Xinje XCPPro project, PLC1: XC2-32 (software 3.3r 2017-11-24)

PROGRAM Ladder

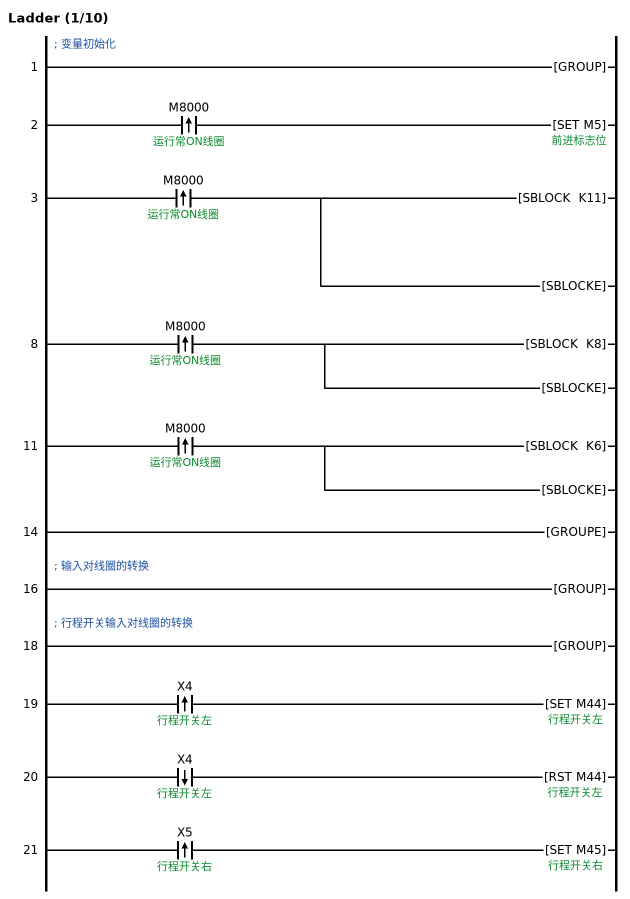
; 变量初始化
GROUP
LDP    M8000	; 运行常ON线圈
SET    M5	; 前进标志位
LDP    M8000	; 运行常ON线圈
SBLOCK K11
SBLOCKE
LDP    M8000	; 运行常ON线圈
SBLOCK K8
SBLOCKE
LDP    M8000	; 运行常ON线圈
SBLOCK K6
SBLOCKE
GROUPE
; 输入对线圈的转换
GROUP
; 行程开关输入对线圈的转换
GROUP
LDP    X4	; 行程开关左
SET    M44	; 行程开关左
LDF    X4	; 行程开关左
RST    M44	; 行程开关左
LDP    X5	; 行程开关右
SET    M45	; 行程开关右

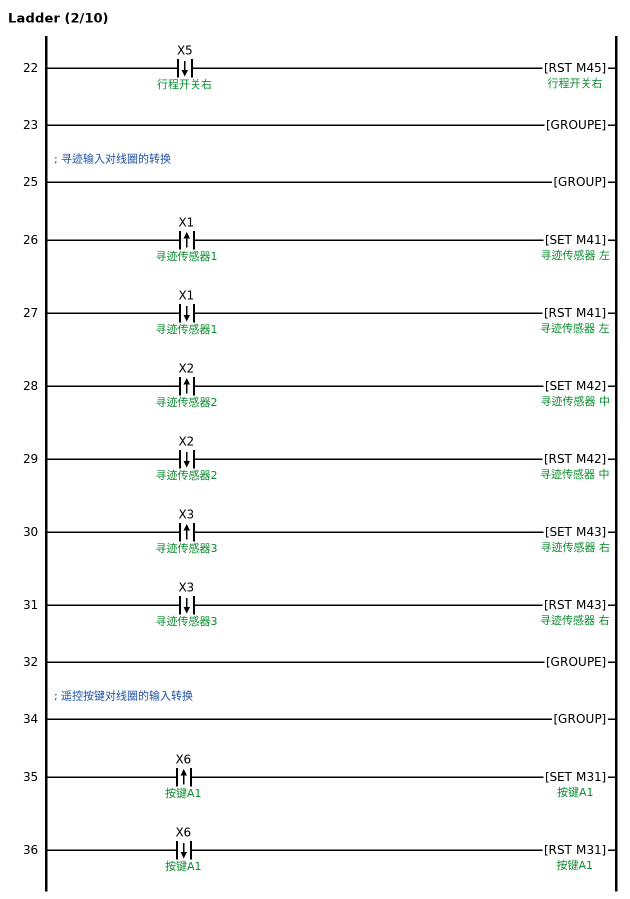
LDF    X5	; 行程开关右
RST    M45	; 行程开关右
GROUPE
; 寻迹输入对线圈的转换
GROUP
LDP    X1	; 寻迹传感器1
SET    M41	; 寻迹传感器 左
LDF    X1	; 寻迹传感器1
RST    M41	; 寻迹传感器 左
LDP    X2	; 寻迹传感器2
SET    M42	; 寻迹传感器 中
LDF    X2	; 寻迹传感器2
RST    M42	; 寻迹传感器 中
LDP    X3	; 寻迹传感器3
SET    M43	; 寻迹传感器 右
LDF    X3	; 寻迹传感器3
RST    M43	; 寻迹传感器 右
GROUPE
; 遥控按键对线圈的输入转换
GROUP
LDP    X6	; 按键A1
SET    M31	; 按键A1
LDF    X6	; 按键A1
RST    M31	; 按键A1

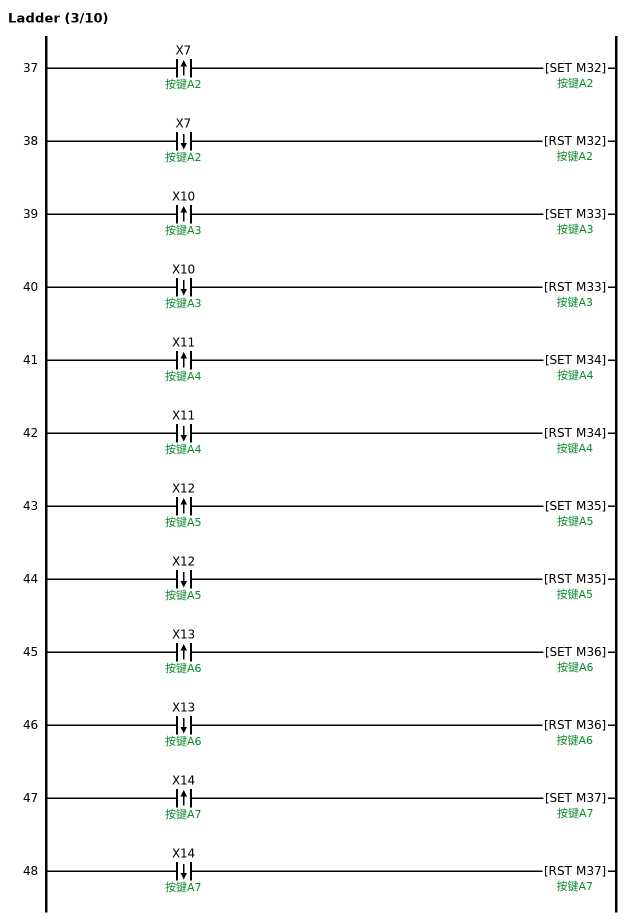
LDP    X7	; 按键A2
SET    M32	; 按键A2
LDF    X7	; 按键A2
RST    M32	; 按键A2
LDP    X10	; 按键A3
SET    M33	; 按键A3
LDF    X10	; 按键A3
RST    M33	; 按键A3
LDP    X11	; 按键A4
SET    M34	; 按键A4
LDF    X11	; 按键A4
RST    M34	; 按键A4
LDP    X12	; 按键A5
SET    M35	; 按键A5
LDF    X12	; 按键A5
RST    M35	; 按键A5
LDP    X13	; 按键A6
SET    M36	; 按键A6
LDF    X13	; 按键A6
RST    M36	; 按键A6
LDP    X14	; 按键A7
SET    M37	; 按键A7
LDF    X14	; 按键A7
RST    M37	; 按键A7

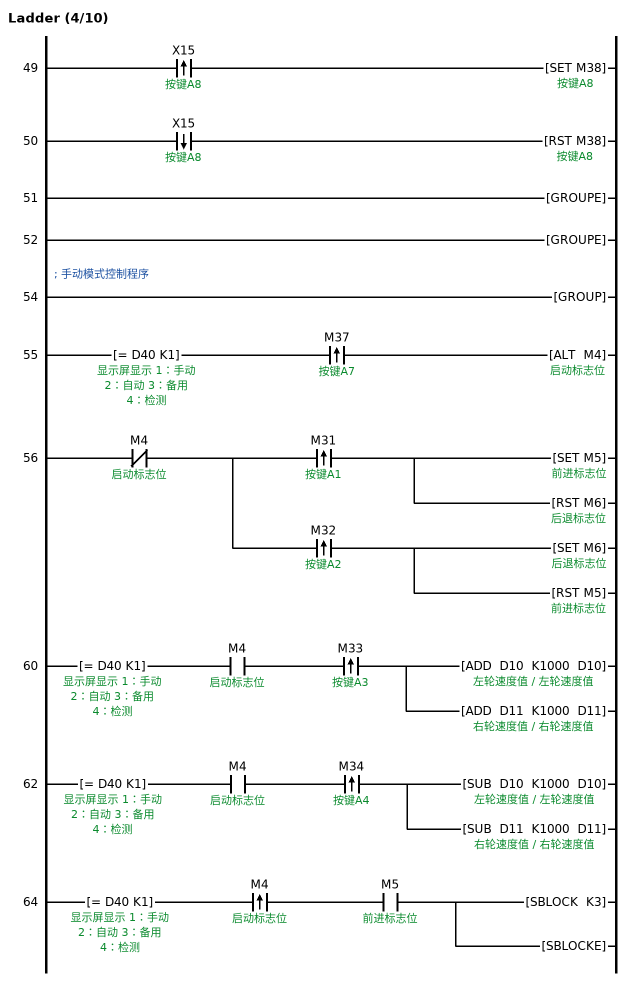
LDP    X15	; 按键A8
SET    M38	; 按键A8
LDF    X15	; 按键A8
RST    M38	; 按键A8
GROUPE
GROUPE
; 手动模式控制程序
GROUP
LD=    D40 K1	; 显示屏显示 1：手动 2：自动 3：备用 4：检测
ANDP   M37	; 按键A7
ALT    M4	; 启动标志位
LDI    M4	; 启动标志位
MPS
ANDP   M31	; 按键A1
SET    M5	; 前进标志位
RST    M6	; 后退标志位
MPP
ANDP   M32	; 按键A2
SET    M6	; 后退标志位
RST    M5	; 前进标志位
LD=    D40 K1	; 显示屏显示 1：手动 2：自动 3：备用 4：检测
AND    M4	; 启动标志位
ANDP   M33	; 按键A3
ADD    D10 K1000 D10	; 左轮速度值 / 左轮速度值
ADD    D11 K1000 D11	; 右轮速度值 / 右轮速度值
LD=    D40 K1	; 显示屏显示 1：手动 2：自动 3：备用 4：检测
AND    M4	; 启动标志位
ANDP   M34	; 按键A4
SUB    D10 K1000 D10	; 左轮速度值 / 左轮速度值
SUB    D11 K1000 D11	; 右轮速度值 / 右轮速度值
LD=    D40 K1	; 显示屏显示 1：手动 2：自动 3：备用 4：检测
ANDP   M4	; 启动标志位
AND    M5	; 前进标志位
SBLOCK K3
SBLOCKE

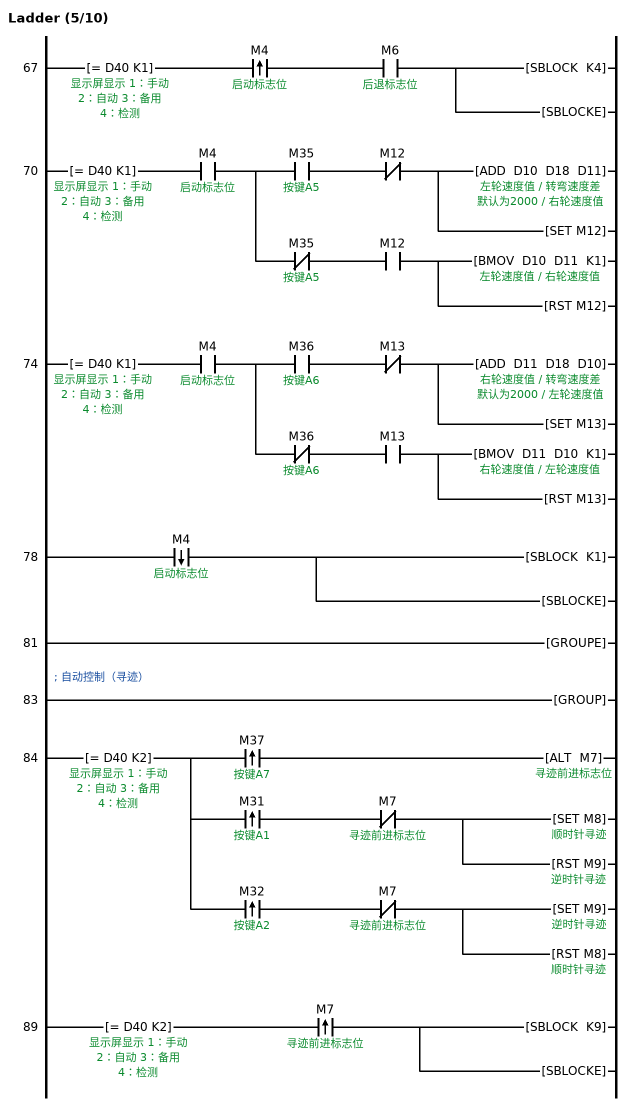
LD=    D40 K1	; 显示屏显示 1：手动 2：自动 3：备用 4：检测
ANDP   M4	; 启动标志位
AND    M6	; 后退标志位
SBLOCK K4
SBLOCKE
LD=    D40 K1	; 显示屏显示 1：手动 2：自动 3：备用 4：检测
AND    M4	; 启动标志位
MPS
AND    M35	; 按键A5
ANI    M12
ADD    D10 D18 D11	; 左轮速度值 / 转弯速度差 默认为2000 / 右轮速度值
SET    M12
MPP
ANI    M35	; 按键A5
AND    M12
BMOV   D10 D11 K1	; 左轮速度值 / 右轮速度值
RST    M12
LD=    D40 K1	; 显示屏显示 1：手动 2：自动 3：备用 4：检测
AND    M4	; 启动标志位
MPS
AND    M36	; 按键A6
ANI    M13
ADD    D11 D18 D10	; 右轮速度值 / 转弯速度差 默认为2000 / 左轮速度值
SET    M13
MPP
ANI    M36	; 按键A6
AND    M13
BMOV   D11 D10 K1	; 右轮速度值 / 左轮速度值
RST    M13
LDF    M4	; 启动标志位
SBLOCK K1
SBLOCKE
GROUPE
; 自动控制（寻迹）
GROUP
LD=    D40 K2	; 显示屏显示 1：手动 2：自动 3：备用 4：检测
MPS
ANDP   M37	; 按键A7
ALT    M7	; 寻迹前进标志位
MRD
ANDP   M31	; 按键A1
ANI    M7	; 寻迹前进标志位
SET    M8	; 顺时针寻迹
RST    M9	; 逆时针寻迹
MPP
ANDP   M32	; 按键A2
ANI    M7	; 寻迹前进标志位
SET    M9	; 逆时针寻迹
RST    M8	; 顺时针寻迹
LD=    D40 K2	; 显示屏显示 1：手动 2：自动 3：备用 4：检测
ANDP   M7	; 寻迹前进标志位
SBLOCK K9
SBLOCKE

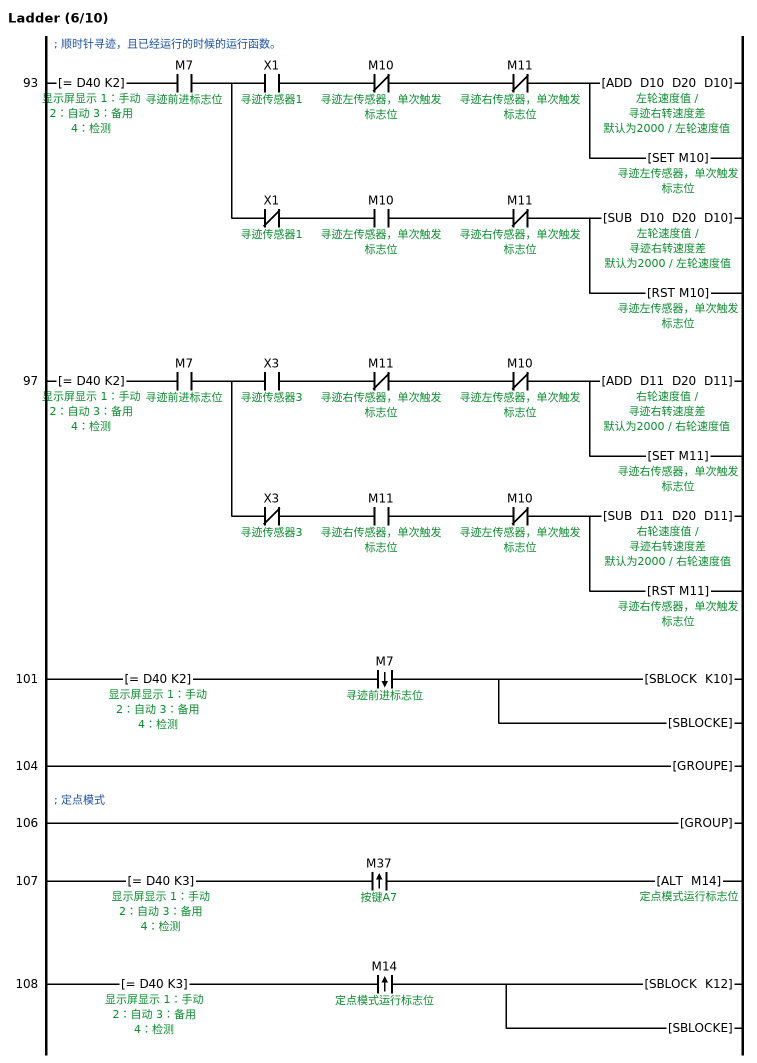
; 顺时针寻迹，且已经运行的时候的运行函数。
LD=    D40 K2	; 显示屏显示 1：手动 2：自动 3：备用 4：检测
AND    M7	; 寻迹前进标志位
MPS
AND    X1	; 寻迹传感器1
ANI    M10	; 寻迹左传感器，单次触发标志位
ANI    M11	; 寻迹右传感器，单次触发标志位
ADD    D10 D20 D10	; 左轮速度值 / 寻迹右转速度差 默认为2000 / 左轮速度值
SET    M10	; 寻迹左传感器，单次触发标志位
MPP
ANI    X1	; 寻迹传感器1
AND    M10	; 寻迹左传感器，单次触发标志位
ANI    M11	; 寻迹右传感器，单次触发标志位
SUB    D10 D20 D10	; 左轮速度值 / 寻迹右转速度差 默认为2000 / 左轮速度值
RST    M10	; 寻迹左传感器，单次触发标志位
LD=    D40 K2	; 显示屏显示 1：手动 2：自动 3：备用 4：检测
AND    M7	; 寻迹前进标志位
MPS
AND    X3	; 寻迹传感器3
ANI    M11	; 寻迹右传感器，单次触发标志位
ANI    M10	; 寻迹左传感器，单次触发标志位
ADD    D11 D20 D11	; 右轮速度值 / 寻迹右转速度差 默认为2000 / 右轮速度值
SET    M11	; 寻迹右传感器，单次触发标志位
MPP
ANI    X3	; 寻迹传感器3
AND    M11	; 寻迹右传感器，单次触发标志位
ANI    M10	; 寻迹左传感器，单次触发标志位
SUB    D11 D20 D11	; 右轮速度值 / 寻迹右转速度差 默认为2000 / 右轮速度值
RST    M11	; 寻迹右传感器，单次触发标志位
LD=    D40 K2	; 显示屏显示 1：手动 2：自动 3：备用 4：检测
ANDF   M7	; 寻迹前进标志位
SBLOCK K10
SBLOCKE
GROUPE
; 定点模式
GROUP
LD=    D40 K3	; 显示屏显示 1：手动 2：自动 3：备用 4：检测
ANDP   M37	; 按键A7
ALT    M14	; 定点模式运行标志位
LD=    D40 K3	; 显示屏显示 1：手动 2：自动 3：备用 4：检测
ANDP   M14	; 定点模式运行标志位
SBLOCK K12
SBLOCKE

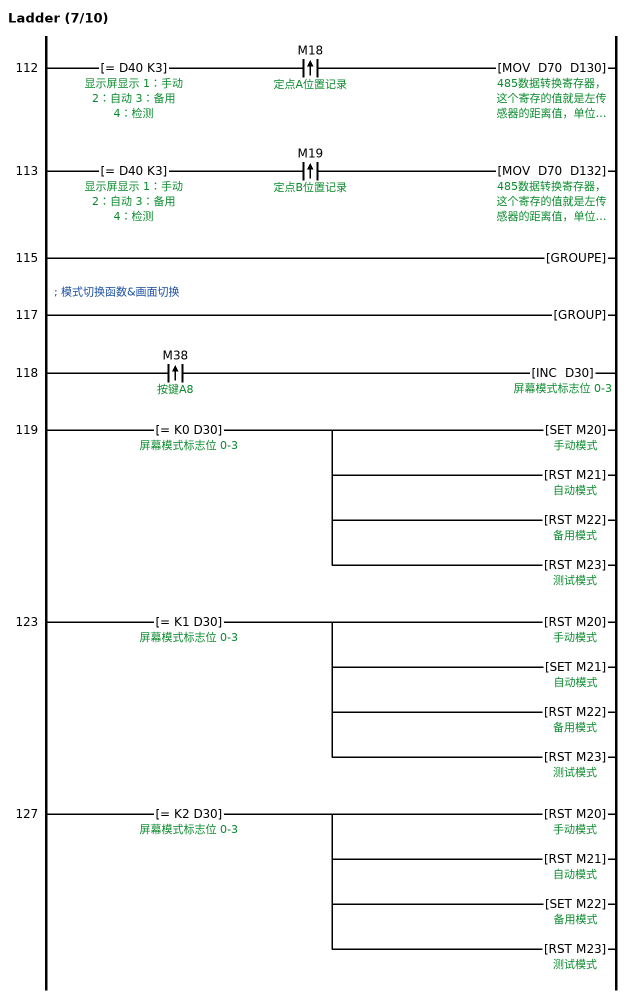
LD=    D40 K3	; 显示屏显示 1：手动 2：自动 3：备用 4：检测
ANDP   M18	; 定点A位置记录
MOV    D70 D130	; 485数据转换寄存器，这个寄存的值就是左传感器的距离值，单位mm / 定点模式A与墙面的距离
LD=    D40 K3	; 显示屏显示 1：手动 2：自动 3：备用 4：检测
ANDP   M19	; 定点B位置记录
MOV    D70 D132	; 485数据转换寄存器，这个寄存的值就是左传感器的距离值，单位mm / 定点模式B与墙面的距离
GROUPE
; 模式切换函数&画面切换
GROUP
LDP    M38	; 按键A8
INC    D30	; 屏幕模式标志位 0-3
LD=    K0 D30	; 屏幕模式标志位 0-3
SET    M20	; 手动模式
RST    M21	; 自动模式
RST    M22	; 备用模式
RST    M23	; 测试模式
LD=    K1 D30	; 屏幕模式标志位 0-3
RST    M20	; 手动模式
SET    M21	; 自动模式
RST    M22	; 备用模式
RST    M23	; 测试模式
LD=    K2 D30	; 屏幕模式标志位 0-3
RST    M20	; 手动模式
RST    M21	; 自动模式
SET    M22	; 备用模式
RST    M23	; 测试模式

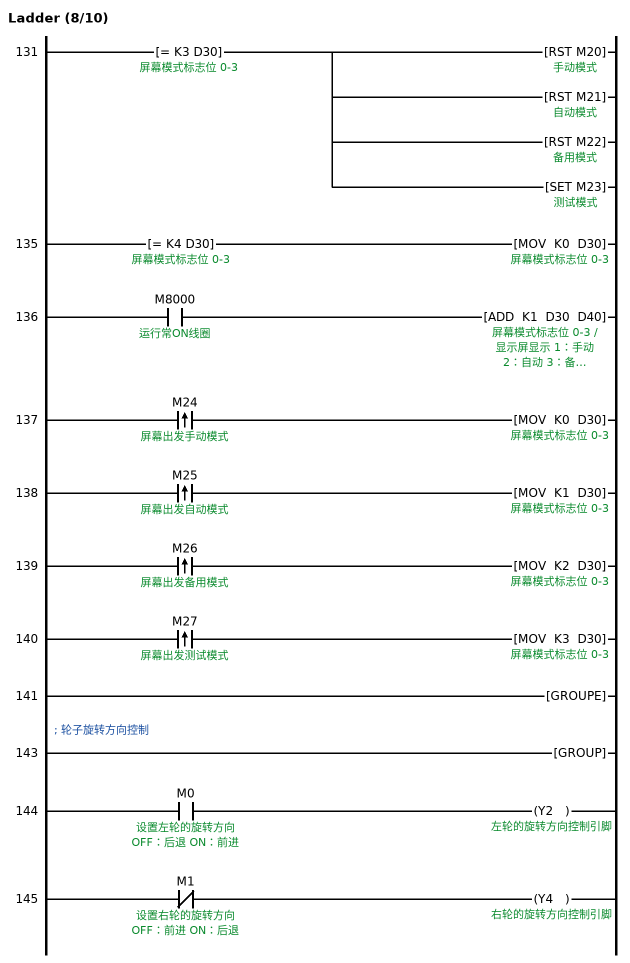
LD=    K3 D30	; 屏幕模式标志位 0-3
RST    M20	; 手动模式
RST    M21	; 自动模式
RST    M22	; 备用模式
SET    M23	; 测试模式
LD=    K4 D30	; 屏幕模式标志位 0-3
MOV    K0 D30	; 屏幕模式标志位 0-3
LD     M8000	; 运行常ON线圈
ADD    K1 D30 D40	; 屏幕模式标志位 0-3 / 显示屏显示 1：手动 2：自动 3：备用 4：检测
LDP    M24	; 屏幕出发手动模式
MOV    K0 D30	; 屏幕模式标志位 0-3
LDP    M25	; 屏幕出发自动模式
MOV    K1 D30	; 屏幕模式标志位 0-3
LDP    M26	; 屏幕出发备用模式
MOV    K2 D30	; 屏幕模式标志位 0-3
LDP    M27	; 屏幕出发测试模式
MOV    K3 D30	; 屏幕模式标志位 0-3
GROUPE
; 轮子旋转方向控制
GROUP
LD     M0	; 设置左轮的旋转方向 OFF：后退 ON：前进 
OUT    Y2	; 左轮的旋转方向控制引脚
LDI    M1	; 设置右轮的旋转方向 OFF：前进 ON：后退
OUT    Y4	; 右轮的旋转方向控制引脚

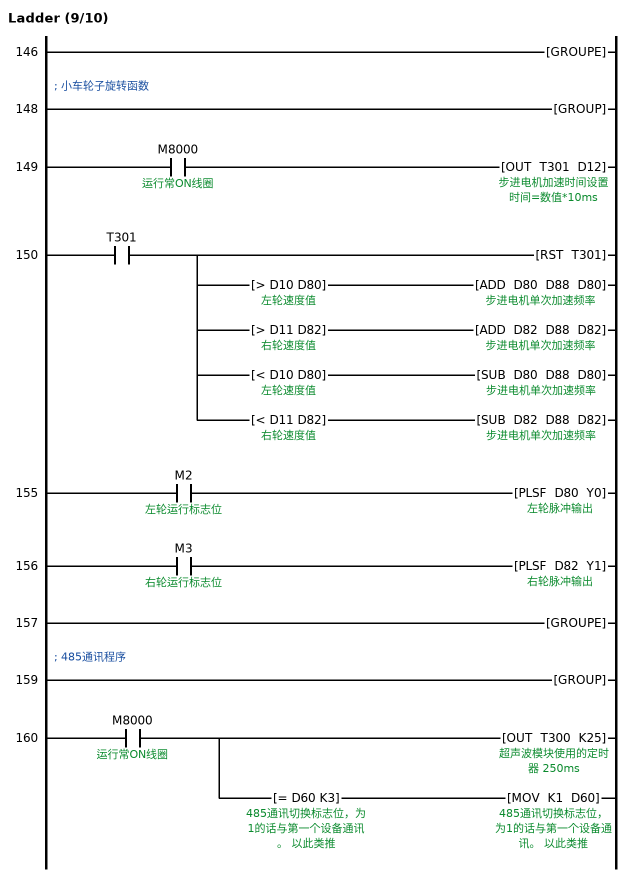
GROUPE
; 小车轮子旋转函数
GROUP
LD     M8000	; 运行常ON线圈
OUT    T301 D12	; 步进电机加速时间设置 时间=数值*10ms
LD     T301
RST    T301
MPS
AND>   D10 D80	; 左轮速度值
ADD    D80 D88 D80	; 步进电机单次加速频率
MRD
AND>   D11 D82	; 右轮速度值
ADD    D82 D88 D82	; 步进电机单次加速频率
MRD
AND<   D10 D80	; 左轮速度值
SUB    D80 D88 D80	; 步进电机单次加速频率
MPP
AND<   D11 D82	; 右轮速度值
SUB    D82 D88 D82	; 步进电机单次加速频率
LD     M2	; 左轮运行标志位
PLSF   D80 Y0	; 左轮脉冲输出
LD     M3	; 右轮运行标志位
PLSF   D82 Y1	; 右轮脉冲输出
GROUPE
; 485通讯程序
GROUP
LD     M8000	; 运行常ON线圈
OUT    T300 K25	; 超声波模块使用的定时器 250ms
AND=   D60 K3	; 485通讯切换标志位，为1的话与第一个设备通讯。 以此类推
MOV    K1 D60	; 485通讯切换标志位，为1的话与第一个设备通讯。 以此类推

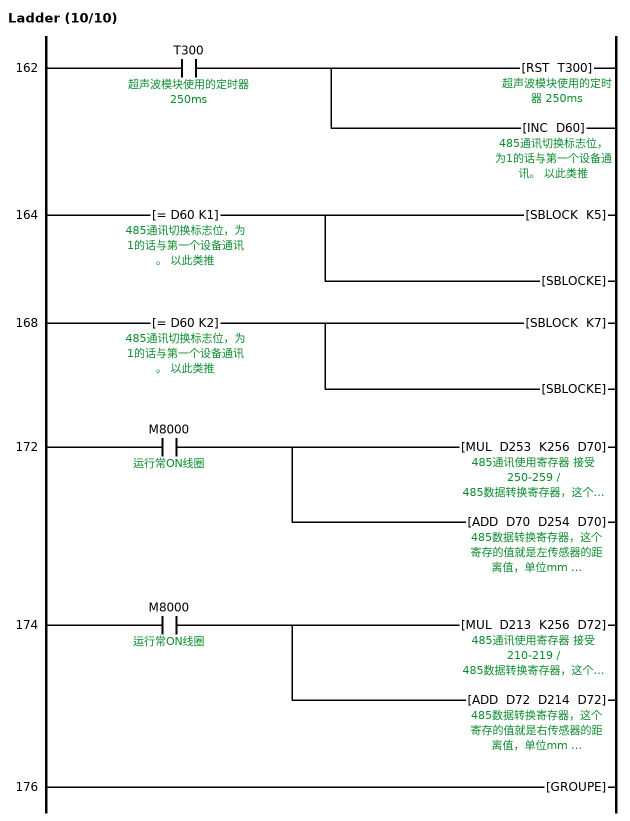
LD     T300	; 超声波模块使用的定时器 250ms
RST    T300	; 超声波模块使用的定时器 250ms
INC    D60	; 485通讯切换标志位，为1的话与第一个设备通讯。 以此类推
LD=    D60 K1	; 485通讯切换标志位，为1的话与第一个设备通讯。 以此类推
SBLOCK K5
SBLOCKE
LD=    D60 K2	; 485通讯切换标志位，为1的话与第一个设备通讯。 以此类推
SBLOCK K7
SBLOCKE
LD     M8000	; 运行常ON线圈
MUL    D253 K256 D70	; 485通讯使用寄存器 接受 250-259 / 485数据转换寄存器，这个寄存的值就是左传感器的距离值，单位mm
ADD    D70 D254 D70	; 485数据转换寄存器，这个寄存的值就是左传感器的距离值，单位mm / 485通讯使用寄存器 接受 250-259 / 485数据转换寄存器，这个寄存的值就是左传感器的距离值，单位mm
LD     M8000	; 运行常ON线圈
MUL    D213 K256 D72	; 485通讯使用寄存器 接受 210-219 / 485数据转换寄存器，这个寄存的值就是右传感器的距离值，单位mm
ADD    D72 D214 D72	; 485数据转换寄存器，这个寄存的值就是右传感器的距离值，单位mm / 485通讯使用寄存器 接受 210-219 / 485数据转换寄存器，这个寄存的值就是右传感器的距离值，单位mm
GROUPE

COMMENTS (devices not used above)
M30	按键A1对应的线圈
D26	小车初始速度 左轮
D28	小车初始速度 右轮
D50	小车运行标志位 0：停止 1：手动前进 2：手动后退
D133	定点的范围差
D134	定点范围差
D200	485通讯使用寄存器 发送data1
D201	485通讯使用寄存器 发送data2
D202	485通讯使用寄存器 发送data3
D203	485通讯使用寄存器 发送data4
D204	485通讯使用寄存器 发送data5
D205	485通讯使用寄存器 发送data6 CRC是206-207
D210	485通讯使用寄存器 接受 210-219
D240	485通讯使用寄存器 发送data1
D241	485通讯使用寄存器 发送data2
D242	485通讯使用寄存器 发送data3
D243	485通讯使用寄存器 发送data4
D244	485通讯使用寄存器 发送data5
D245	485通讯使用寄存器 发送data6 CRC是206-207
D250	485通讯使用寄存器 接受 250-259

SBLOCK K1	; 小车停止
  ; 命令语列表
  RST M2
  RST M3
  RST M1
  RST M0
  MOV K0 D10
  MOV K0 D11

SBLOCK K2	; 顺序功能块2
  ; 命令语列表
  SET M2
  SET M3
  SET M1
  SET M0
  MOV K1000 D10
  MOV K1000 D11

SBLOCK K3	; 小车的低速前进
  ; 命令语列表
  SET M2
  SET M3
  SET M1
  SET M0
  MOV K1000 D10
  MOV K1000 D11

SBLOCK K4	; 小车的低速后退
  ; 命令语列表
  SET M2
  SET M3
  RST M1
  RST M0
  MOV K1000 D10
  MOV K1000 D11

SBLOCK K5	; 超声波1收发指令
  ; SEND
  T_COMM
  SEND
  ; InstType=T_COMM, IsUserInst=false, PLCAddr=D200, ComNum=K3, BufferCount=8, Reg=D200, RegByteCount=6, RegByteCount=0, CheckReg=D200, CheckLen=6, GUID=69af5672-a25c-46f3-9e3d-716bfc8745a2
  ; REV
  T_COMM
  RCV
  ; InstType=T_COMM, IsUserInst=false, PLCAddr=D210, ComNum=K3, BufferCount=8, Reg=D210, RegByteCount=10, GUID=67083cb6-353a-4d1b-a49b-9335a17586a7

SBLOCK K6	; 初始化寄存器_485SEND1
  ; 命令语列表
  MOV K1 D200
  MOV K3 D201
  MOV K1 D202
  MOV K1 D203
  MOV K0 D204
  MOV K1 D205

SBLOCK K7	; 超声波2收发指令
  ; SEND2
  T_COMM
  SEND
  ; InstType=T_COMM, IsUserInst=false, PLCAddr=D240, ComNum=K3, BufferCount=8, Reg=D240, RegByteCount=6, RegByteCount=0, CheckReg=D240, CheckLen=6, GUID=c498a6d9-c5eb-440f-ad17-3bc66fdd4bec
  ; REV2
  T_COMM
  RCV
  ; InstType=T_COMM, IsUserInst=false, PLCAddr=D250, ComNum=K3, BufferCount=8, Reg=D250, RegByteCount=10, GUID=fb04215a-2533-426a-b545-081527f59ed3

SBLOCK K8	; 初始化寄存器_485SEND2
  ; 命令语列表
  MOV K2 D240
  MOV K3 D241
  MOV K1 D242
  MOV K1 D243
  MOV K0 D244
  MOV K1 D245

SBLOCK K9	; 寻迹小车前进
  ; 命令语列表
  SET M2
  SET M3
  SET M1
  SET M0
  MOV D26 D10
  MOV D28 D11

SBLOCK K10	; 寻迹小车停止
  ; 命令语列表
  RST M2
  RST M3
  RST M1
  RST M0
  MOV K00 D10
  MOV K00 D11

SBLOCK K11	; 变量初始化
  ; 变量初始化
  MOV K3000 D26
  MOV K3000 D28
  MOV K0 D8170
  MOV K0 D8173
  MOV K2000 D100
  MOV K30000 D101
  MOV K2000 D110
  MOV K30000 D111
  MOV K30000 D105
  MOV K30000 D115
  PLSMV K0 Y0
  PLSMV K0 Y1
  MOV K5 D12
  MOV K5000 D18
  MOV K5000 D20
  ; 定点模式初始化
  MOV K0 D130
  MOV K0 D132
  MOV K30 D134
  MOV K0 D135
  MOV K0 D136
  MOV K0 D139
  ; 单次步进电机加减速值
  MOV K500 D88

SBLOCK K12	; 定点模式起始
  ; 小车前进
  SET M2
  SET M3
  SET M1
  SET M0
  MOV K1000 D10
  MOV K1000 D11

C FUNCTION BLOCK car_run.fcb
/*************************************************************************
   FunctionBlockName:  CAR_RUN
   Version:            1.0.0
   Author:             赵海行
   UpdateTime:         2023/6/13 9:49:36
   Comment:            
			小车的底层运行标志位设置
**************************************************************************/
void CAR_RUN( WORD W , BIT B )
{

	B[0]=1;
	B[1]=1;
	B[2]=1;
	B[3]=1;

}

C FUNCTION BLOCK tca.fcb
/* 圆面积的计算【半径为整数】
半径数据输入(整数)： W[0]
圆面积值输出(浮点数):FW[2]
例:
TCA D0 M0
半径:   D0=2
圆面积：F(D2,D3)=_PI*D0*D0
=π*2*2
结果:   4π */
/*************************************************************************
   FunctionBlockName:  TCA
   Version:            1.0.0
   Author:             无锡信捷电气有限公司
   UpdateTime:         2010-4-21 21:03:31
   Comment:            
			圆面积的计算【半径为整数】            
			
			
			半径数据输入(整数)： W[0]
      圆面积值输出(浮点数):FW[2]
			例:
			TCA D0 M0
			
			半径:   D0=2  
			圆面积：F(D2,D3)=_PI*D0*D0
			                =π*2*2
			结果:   4π
			   
**************************************************************************/
void TCA( WORD W , BIT B )
{
   FW[2]=W[0]*W[0]*_PI;
 }